Staubli VAL3: TYPELEN.pgx

public program typeLen(num x_nX, num x_nY, string x_sMessage, num x_nLength)
begin
  //-----------------------------------------------------------------------
  //Header begin
  //Description of program
  //  Displays one message to pX column and pY Line.
  //  If the length of the message is less than x_nLen, the characters are replaced
  //  by spaces otherwise the message will be truncated.
  //
  //Input parameters
  //  num x_nX :
  //    role : cursor column
  //  num x_nY :
  //    role : cursor row
  //  string x_sMessage :
  //    role : message that you want to display
  //  num x_nLength :
  //    role : max length of the message
  //
  //Example
  //  call typeLen(2,5,"Hello",10)
  //
  //History
  //  Creation : 28-04-08 - f.Rob
  //Header end
  //-----------------------------------------------------------------------
  call strlength(x_sMessage,x_nLength)
  call type(x_nX,x_nY,x_sMessage)
end
